FUNCTION F_CalcSum3DimArray : LREAL
VAR_IN_OUT
	arrData		: ARRAY[*, *, *] OF LREAL;
END_VAR
VAR
	nIndex1, nIndex2, nIndex3	: DINT;
END_VAR

F_CalcSum3DimArray := 0;
FOR nIndex1 := LOWER_BOUND(arrData, 1) TO UPPER_BOUND(arrData, 1) DO
	FOR nIndex2 := LOWER_BOUND(arrData, 2) TO UPPER_BOUND(arrData, 2) DO
		FOR nIndex3 := LOWER_BOUND(arrData, 3) TO UPPER_BOUND(arrData, 3) DO
			F_CalcSum3DimArray := F_CalcSum3DimArray + arrData[nIndex1, nIndex2, nIndex3];
		END_FOR
	END_FOR
END_FOR

END_FUNCTION

(* stored: Version 1.1.0.1, ProductVersion 3.1.4019.2
   POU F_CalcSum3DimArray: Id {c945c67e-59b3-4261-bd04-93c0970e1651}, SpecialFunc None *)
